// SIMATIC S7-200 project (STEP 7-Micro/WIN), CPU 224 REL 01.21

ORGANIZATION_BLOCK 主程序:OB1
TITLE=程序注释
BEGIN
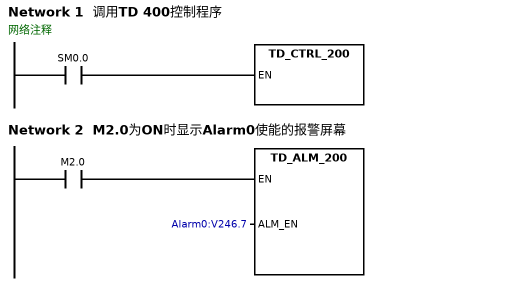
Network 1 // 调用TD 400控制程序
// 网络注释
LD     SM0.0
CALL   TD_CTRL_200:SBR1
Network 2 // M2.0为ON时显示Alarm0使能的报警屏幕
LD     M2.0
CALL   TD_ALM_200:SBR2, Alarm0:V246.7
END_ORGANIZATION_BLOCK

// SBR1: protected block, not included

// SBR2: protected block, not included

// (further data pages could not be read)
